// TIA Portal V20 export
// export: Created 2025-12-01T14:57:21.0848752Z, ExportSetting None, DisplayName Totally Integrated Automation Portal, DisplayVersion V20 Update 3, DisplayName TIA Portal Openness, DisplayVersion V20 Update 3, DisplayName TIA Portal Version Control Interface, DisplayVersion V20 Update 3, DisplayName STEP 7 Professional, DisplayVersion V20 Update 3, DisplayName STEP 7 Safety, DisplayVersion V20 Update 2, DisplayName WinCC Basic/Comfort/Advanced, DisplayVersion V20 Update 3, DisplayName WinCC Professional, DisplayVersion V20 Update 3, DisplayName WinCC Unified, DisplayVersion V20 Update 3
DATA_BLOCK "DB2130_DB_BarrSeg1"   // DB2130, F_DB
FAMILY : FPRI085d
VERSION : 0.0
// stored: AutoNumber false, InstanceOfName FB2141_F_BarreraSeguridad, InstanceOfType FB
"FB2141_F_BarreraSeguridad"
   // VAR_INPUT
   //    NumBarrera : Int;
   //    Modo_Ventana : Bool;
   //    MS_11 : Bool;
   //    MS_12 : Bool;
   //    MS_21 : Bool;
   //    MS_22 : Bool;
   //    Potencia_Desactivada : Bool;
   //    Barrera : Bool;
   //    ENABLE : Bool;
   //    ACK : Bool;
   //    DISC_TIME_1 : Time;
   //    DISC_TIME_2 : Time;
   //    TIME_MAX : Time;
   //    TIME_Ventana_INI : Time;
   //    TIME_Ventana_FIN : Time;
   // END_VAR
   // VAR_OUTPUT
   //    Q : Bool;
   //    MUTING_LAMP : Bool;
   //    ACK_REQ : Bool;
   //    FAULT : Bool;
   // END_VAR
   // VAR
   //    F_MUT_P { S7_SetPoint := 'True'} : MUT_P;
   //    F_TON_INI { S7_SetPoint := 'True'} : TON;
   //    F_TON_FIN { S7_SetPoint := 'True'} : TON;
   //    Ventana_Q : Bool;
   // END_VAR
BEGIN
END_DATA_BLOCK
